# B&R Automation Studio project TD52 (part 142)

#### lGEN2diag.typ
```iecst
TYPE

   DiagActiveBus : STRUCT
        DiagOn : BOOL; (**)
        DiagOnInTransient : BOOL; (**)
        LEANOXErrSettled : BOOL; (**)
        NoTooStrongWGMove : BOOL; (**)
        NoTransient : BOOL; (**)
        NoExtDist : BOOL; (**)
        NoVoltTrans : BOOL; (**)
        GCBMCBsettled : BOOL; (**)
        GridP : BOOL; (**)
        DiagBitmask : DINT; (**)
        NoMinLoad : BOOL; (**)
        TexhSettledAfterRamp : BOOL; (**)
        NoGasMixingTrans : BOOL; (**)
    END_STRUCT;

   tGEN2FDebug : STRUCT
        LambdaCmd : REAL; (*lambda command [-]*)
        y_f : REAL; (*filtered value of y*)
        Residual : REAL; (*high pass filtered lambda (= gradient)*)
        Thrsh : REAL; (*the actual threshold (after scaling)*)
        DiagActive : BOOL; (*diagnosis activated*)
        FaultLambdaOnly : BOOL; (*fault detected based only on lambda gradient (WITHOUT deactivation logic)*)
        ResLambdaOnly : REAL; (*high pass filtered lambda signal (after lambda has been lowpass filtered)*)
        ResLambdaITP : REAL; (*high pass filtered lambda signal due to ITP change (after lambda est. has been lowpass filtered)*)
        ResLambdaEst : REAL; (*high pass filtered estimated lambda signal (after lambda est. has been lowpass filtered)*)
        LambdaEst : REAL; (*estimated lambda (via lookup table) dependent on p2s*)
        LEANOXErr : REAL; (*internally calculated LEANOX error [bar]*)
        TexhAvg : REAL; (*exhaust temperature [°C] (avg.) calculated via the mean value*)
        TexhMin : REAL; (*exhaust temperature [°C] (min.)*)
        GasMixing_RatioHP : REAL; (*high pass filtered gas mixing ratio*)
        DeltaTexhAllowed : REAL; (*max. allowed rise in avg. exhaust temp. [°C] used for fault detection (after scaling)*)
        tDiagActiveBus : DiagActiveBus; (*struct to check which component of the activation logic is on*)
    END_STRUCT;

   tGEN2FIn : STRUCT
        LambdaCmd : REAL; (*lambda command [-]*)
        Lambda_ss : REAL; (*steady state lambda [-]*)
        Reset : BOOL; (*reset of filter blocks*)
        Pset_WR_norm : REAL; (*power reference without a ramp [p.u.]*)
        Pset_norm : REAL; (*power reference trajectory [p.u.]*)
        bExt_dist : BOOL; (*TRUE --> external disturbance*)
        Texh : ARRAY[0..24] OF REAL; (*exhaust temperatures (cylinder specific)*)
        p2s : REAL; (*p2s [bar]*)
        p2sCmd : REAL; (*p2s command (LEANOX) [bar]*)
        posWG_norm : REAL; (*waste-gate position [p.u.] 0...1*)
        WGM_reset : BOOL; (*reset bit for the wastegate monitoring part*)
        LEANOXErrorFiltReset : BOOL; (*reset bit for the lowpass used to filter p2s in the LEANOX error settling detection*)
        bVltg_reset : BOOL; (*reset bit for the voltage monitoring part*)
        U_L1L2_norm : REAL; (*concatenated voltage L1L2 [p.u.]*)
        U_L2L3_norm : REAL; (*concatenated voltage L2L3 [p.u.]*)
        U_L3L1_norm : REAL; (*concatenated voltage L1L2 [p.u.]*)
        Man_Cond_On : BOOL; (*manual override to set the diagnosis to ON*)
        bGCBON : BOOL; (*generator circuit breaker closed information*)
        bMCBON : BOOL; (*main circuit breaker closed information*)
        bPTransDetReset : BOOL; (*reset bit for the transient monitoring part*)
        bAllowDetInTrans : BOOL; (*allow detection during ramps (if LEANOX error is small enough)*)
        bTexhSettled_reset : BOOL; (*reset bit for Texh settled detection (after power ramps)*)
        rGasMixing_Ratio : REAL; (*gas mixing ratio [0 - 100 percent]*)
        bGasMixing_reset : BOOL; (*reset bit for gas mixing settled detection*)
        bFileOnlyInTrans : BOOL; (*write files only during power ramps (only if detection is allowed during ramps)*)
        rITPmean : REAL; (*mean ignition timing point [°CA]*)
    END_STRUCT;

   tGEN2FOut : STRUCT
        FrictionFault : BOOL; (*fault detected based on (negative) lambda gradient and (positive) exh. temp. gradient*)
        FrictionFaultInTransient : BOOL; (*fault detected based on (negative) lambda gradient and (positive) exh. temp. gradient; fault in transient detected (only for writing files at the moment!)*)
    END_STRUCT;

   tGEN2FParameter : STRUCT
        TrshPsetDev : REAL; (*threshold value for power set point deviation [p.u.]*)
        TrshPsetStat : REAL; (*threshold value for steady state detection [p.u.]*)
        TconstPsetStat : REAL; (*timeconstant for steady state detection*)
        TrshLoad : REAL; (*threshold value for load level (related to the set power point) [p.u.]*)
        TConstLP : REAL; (*time constant [s] for the lambda lowpass filter*)
        TConstHP : REAL; (*time constant [s] for the lambda highpass filter (situated after the lowpass)*)
        ITPmeanScaling : REAL; (*scaling for the mean ITP to estimate a lambda change*)
        FaultThrshLambda : REAL; (*threshold value for lambda fault detection*)
        ThrshScale : REAL; (*scaling of the threshold value for lambda fault detection [p.u.]*)
        TPulseLambdaFault : REAL; (*minimum time [s] a lambda fault pulse is provided for further detection (exh. temp.)*)
        NCyl : DINT; (*number of cylinders*)
        DeltaTexhAllowed : REAL; (*max. allowed rise in avg. exhaust temp. used for fault detection*)
        TexhPlausibleMin : REAL; (*min. exhaust temperature which is considered plausible (to exclude faulty sensors)*)
        TexhPlausibleMax : REAL; (*max. exhaust temperature which is considered plausible (to exclude faulty sensors)*)
        WGM_FaultThrsh : REAL; (*wastegate monitoring fault threshold*)
        WGM_Tconst : REAL; (*wastegate monitoring time constant [sec]*)
        LEANOXErrorTconst : REAL; (*time constant [s] for filtering p2s in LEANOX error calculation*)
        LEANOXErrorThrsh : REAL; (*threshold for leanox error (diagnosis gets active if the error is smaller than this threshold)*)
        Vltg_FaultThrsh : REAL; (*voltage monitoring fault threshold*)
        Vltg_Tconst : REAL; (*voltage monitoring time constant [sec]*)
        MonitoringDelay : REAL; (*global monitoring time delay (used for all activation logic pars) [sec]*)
        TexhSettledThrsh : REAL; (*threshold for exhaust temperature settled detection*)
        TexhSettledTConstLP : REAL; (*time constant [s] for the Texh lowpass filter -> settled detection*)
        TexhSettledTConstHP : REAL; (*time constant [s] for the Texh highpass filter (situated after the lowpass) -> settled detection*)
        TexhSettledMaxTD : REAL; (*max. time [s] after a power ramp after which the exhaust temperature is considered settled (even if the filter does not suggest this!)*)
        bGasMixingEnDet : BOOL; (*enable gas mixing transient detection*)
        GasMixingThrsh : REAL; (*threshold for gas mixing transient detection*)
        GasMixingTconstLP : REAL; (*time constant [s] for gas mixing transient detection lowpass*)
        GasMixingTconstHP : REAL; (*time constant [s] for gas mixing transient detection highpass*)
    END_STRUCT;
END_TYPE
TYPE
rtB_TOF_G2Fdiag : STRUCT
	LogicalOperator1 : BOOL;
END_STRUCT;
rtDW_TOF_G2Fdiag : STRUCT
	DiscreteTimeIntegrator_DSTATE : LREAL;
	DiscreteTimeIntegrator_PrevRese : SINT;
	DiscreteTimeIntegrator_IC_LOADI : USINT;
END_STRUCT;
rtB_TON_G2Fdiag : STRUCT
	LogicalOperator3 : BOOL;
END_STRUCT;
rtDW_TON_G2Fdiag : STRUCT
	DiscreteTimeIntegrator_DSTATE : REAL;
	DiscreteTimeIntegrator_PrevRese : SINT;
END_STRUCT;
rtB_TP_G2Fdiag : STRUCT
	Merge : LREAL;
	LogicalOperator1 : BOOL;
END_STRUCT;
rtDW_TP_G2Fdiag : STRUCT
	DelayInput2_DSTATE : LREAL;
	UnitDelay2_DSTATE : BOOL;
END_STRUCT;
BlockIO_G2Fdiag : STRUCT
	BusInput1 : tGEN2FIn;
	BusInput : tGEN2FParameter;
	UnitDelay : UDINT;
	TP1 : rtB_TP_G2Fdiag;
	TP : rtB_TP_G2Fdiag;
	TON_n : rtB_TON_G2Fdiag;
	TON_i : rtB_TON_G2Fdiag;
	TON1 : rtB_TON_G2Fdiag;
	TON_e : rtB_TON_G2Fdiag;
	TOF_o : rtB_TOF_G2Fdiag;
	TOF_h : rtB_TOF_G2Fdiag;
	TON : rtB_TON_G2Fdiag;
	TON_j : rtB_TON_G2Fdiag;
	TON_k : rtB_TON_G2Fdiag;
	TOF : rtB_TOF_G2Fdiag;
END_STRUCT;
D_Work_G2Fdiag : STRUCT
	DiscreteTimeIntegrator_DSTATE : REAL;
	DiscreteTimeIntegrator_DSTATE_k : REAL;
	DiscreteTimeIntegrator_DSTATE_h : REAL;
	DiscreteTimeIntegrator_DSTATE_c : REAL;
	DiscreteTimeIntegrator_DSTATE_p : REAL;
	DiscreteTimeIntegrator_DSTATE_e : REAL;
	DiscreteTimeIntegrator_DSTAT_hv : REAL;
	DiscreteTimeIntegrator_DSTATE_j : REAL;
	DiscreteTimeIntegrator_DSTATE_n : REAL;
	DiscreteTimeIntegrator_DSTATE_o : ARRAY[0..2] OF REAL;
	DiscreteTimeIntegrator_DSTAT_jn : ARRAY[0..2] OF REAL;
	DiscreteTimeIntegrator_DSTATE_a : ARRAY[0..2] OF REAL;
	DiscreteTimeIntegrator_DSTATE_d : ARRAY[0..2] OF REAL;
	DiscreteTimeIntegrator_DSTATE_i : REAL;
	UnitDelay_DSTATE : UDINT;
	Texh_scalar_1 : REAL;
	Texh_min_1 : REAL;
	Texh_scalar_1_f : REAL;
	Texh_min_1_p : REAL;
	DelayInput1_DSTATE : BOOL;
	DelayInput1_DSTATE_e : BOOL;
	DelayInput1_DSTATE_m : BOOL;
	DelayInput1_DSTATE_l : BOOL;
	Delay_DSTATE : BOOL;
	DelayInput1_DSTATE_i : BOOL;
	DelayInput1_DSTATE_n : BOOL;
	DelayInput1_DSTATE_p : BOOL;
	DelayInput1_DSTATE_p3 : BOOL;
	DiscreteTimeIntegrator_PrevRese : SINT;
	DiscreteTimeIntegrator_PrevRe_e : SINT;
	DiscreteTimeIntegrator_PrevRe_j : SINT;
	DiscreteTimeIntegrator_PrevRe_f : SINT;
	DiscreteTimeIntegrator_PrevRe_p : SINT;
	DiscreteTimeIntegrator_PrevR_jm : SINT;
	DiscreteTimeIntegrator_PrevRe_n : SINT;
	DiscreteTimeIntegrator_PrevR_ji : SINT;
	DiscreteTimeIntegrator_PrevR_nv : SINT;
	DiscreteTimeIntegrator_PrevRe_d : SINT;
	DiscreteTimeIntegrator_PrevR_do : SINT;
	DiscreteTimeIntegrator_PrevRe_m : SINT;
	DiscreteTimeIntegrator_PrevRe_a : SINT;
	DiscreteTimeIntegrator_PrevR_ah : SINT;
	DiscreteTimeIntegrator_IC_LOADI : USINT;
	DiscreteTimeIntegrator_IC_LOA_c : USINT;
	DiscreteTimeIntegrator_IC_LOA_b : USINT;
	DiscreteTimeIntegrator_IC_LOA_g : USINT;
	DiscreteTimeIntegrator_IC_LOA_p : USINT;
	DiscreteTimeIntegrator_IC_LOA_o : USINT;
	DiscreteTimeIntegrator_IC_LO_cl : USINT;
	DiscreteTimeIntegrator_IC_LO_ps : USINT;
	DiscreteTimeIntegrator_IC_LOA_h : USINT;
	DiscreteTimeIntegrator_IC_LO_pk : USINT;
	DiscreteTimeIntegrator_IC_LO_c0 : USINT;
	DiscreteTimeIntegrator_IC_LOA_j : USINT;
	DiscreteTimeIntegrator_IC_LOA_e : USINT;
	DiscreteTimeIntegrator_IC_LO_gt : USINT;
	Texh_scalar_1_not_empty : BOOL;
	Texh_scalar_1_not_empty_d : BOOL;
	bSettlingPhase : BOOL;
	TexhSettledAfterRamp_persistent : BOOL;
	TP1 : rtDW_TP_G2Fdiag;
	TP : rtDW_TP_G2Fdiag;
	TON_n : rtDW_TON_G2Fdiag;
	TON_i : rtDW_TON_G2Fdiag;
	TON1 : rtDW_TON_G2Fdiag;
	TON_e : rtDW_TON_G2Fdiag;
	TOF_o : rtDW_TOF_G2Fdiag;
	TOF_h : rtDW_TOF_G2Fdiag;
	TON : rtDW_TON_G2Fdiag;
	TON_j : rtDW_TON_G2Fdiag;
	TON_k : rtDW_TON_G2Fdiag;
	TOF : rtDW_TOF_G2Fdiag;
END_STRUCT;
ExternalInputs_G2Fdiag : STRUCT
	IN : tGEN2FIn;
	para : tGEN2FParameter;
END_STRUCT;
ExternalOutputs_G2Fdiag : STRUCT
	OUT : tGEN2FOut;
	dbg : tGEN2FDebug;
END_STRUCT;
END_TYPE
```

#### G2Fdiag.h
```c
/********************************************************************
 * COPYRIGHT -- Bernecker + Rainer Industrie-Elektronik Ges.m.b.H.
 ********************************************************************
 * Program: G2Fdiag
 * File: G2Fdiag.h
 * Author: 106003773
 * Created: Wed Apr 20 16:09:39 2016
 ********************************************************************
 * Header for program G2Fdiag
 ********************************************************************
 * Generated with B&R Automation Studio Target for Simulink V4.2
 * (ERT based)
 ********************************************************************/

#ifndef RTW_HEADER_G2Fdiag_h_
#define RTW_HEADER_G2Fdiag_h_
#ifndef G2Fdiag_COMMON_INCLUDES_
# define G2Fdiag_COMMON_INCLUDES_
#include <math.h>
#include "rtwtypes.h"
#include "rtw_continuous.h"
#include "rtw_solver.h"
#endif                                 /* G2Fdiag_COMMON_INCLUDES_ */

#include "G2Fdiag_types.h"
#include "lGEN2diag.h"

/* Macros for accessing real-time model data structure */
#ifndef rtmGetErrorStatus
# define rtmGetErrorStatus(rtm)        ((void*) 0)
#endif

#ifndef rtmSetErrorStatus
# define rtmSetErrorStatus(rtm, val)   ((void) 0)
#endif

#ifndef rtmGetStopRequested
# define rtmGetStopRequested(rtm)      ((void*) 0)
#endif

#ifndef MIN
#define MIN(a,b)                       ((a) < (b) ? (a) : (b))
#endif

#ifndef MAX
#define MAX(a,b)                       ((a) > (b) ? (a) : (b))
#endif

/* Block signals for system '<S7>/TOF' */

/* Block states (auto storage) for system '<S7>/TOF' */

/* Block signals for system '<S8>/TON' */

/* Block states (auto storage) for system '<S8>/TON' */

/* Block signals for system '<S6>/TP' */

/* Block states (auto storage) for system '<S6>/TP' */

/* Block signals (auto storage) */

/* Block states (auto storage) for system '<Root>' */

/* External inputs (root inport signals with auto storage) */

/* External outputs (root outports fed by signals with auto storage) */

/* Block signals (auto storage) */
extern BlockIO_G2Fdiag G2Fdiag_B;

/* Block states (auto storage) */
extern D_Work_G2Fdiag G2Fdiag_DWork;

/* External inputs (root inport signals with auto storage) */
extern ExternalInputs_G2Fdiag G2Fdiag_U;

/* External outputs (root outports fed by signals with auto storage) */
extern ExternalOutputs_G2Fdiag G2Fdiag_Y;

/* Model entry point functions */
extern void G2Fdiag_initialize(struct fGEN2diag* inst);
extern void G2Fdiag_step(struct fGEN2diag* inst);
extern void G2Fdiag_terminate(struct fGEN2diag* inst);

/*-
 * The generated code includes comments that allow you to trace directly
 * back to the appropriate location in the model.  The basic format
 * is <system>/block_name, where system is the system number (uniquely
 * assigned by Simulink) and block_name is the name of the block.
 *
 * Use the MATLAB hilite_system command to trace the generated code back
 * to the model.  For example,
 *
 * hilite_system('<S3>')    - opens system 3
 * hilite_system('<S3>/Kp') - opens and selects block Kp which resides in S3
 *
 * Here is the system hierarchy for this model
 *
 * '<Root>' : 'G2Fdiag'
 * '<S1>'   : 'G2Fdiag/Environment Controller'
 * '<S2>'   : 'G2Fdiag/Environment Controller1'
 * '<S3>'   : 'G2Fdiag/GEN2_Friction_Detection'
 * '<S4>'   : 'G2Fdiag/Info'
 * '<S5>'   : 'G2Fdiag/GEN2_Friction_Detection/DiagActivLogic'
 * '<S6>'   : 'G2Fdiag/GEN2_Friction_Detection/Fault Detection'
 * '<S7>'   : 'G2Fdiag/GEN2_Friction_Detection/DiagActivLogic/Exteternal disturbance'
 * '<S8>'   : 'G2Fdiag/GEN2_Friction_Detection/DiagActivLogic/GBC and MBC monitoring'
 * '<S9>'   : 'G2Fdiag/GEN2_Friction_Detection/DiagActivLogic/GasMixingTransient'
 * '<S10>'  : 'G2Fdiag/GEN2_Friction_Detection/DiagActivLogic/LEANOX error monitoring'
 * '<S11>'  : 'G2Fdiag/GEN2_Friction_Detection/DiagActivLogic/Min Load Detection'
 * '<S12>'  : 'G2Fdiag/GEN2_Friction_Detection/DiagActivLogic/Power ramp detection'
 * '<S13>'  : 'G2Fdiag/GEN2_Friction_Detection/DiagActivLogic/Texh settled after power ramp'
 * '<S14>'  : 'G2Fdiag/GEN2_Friction_Detection/DiagActivLogic/Voltage monitoring'
 * '<S15>'  : 'G2Fdiag/GEN2_Friction_Detection/DiagActivLogic/Wastegate monitoring'
 * '<S16>'  : 'G2Fdiag/GEN2_Friction_Detection/DiagActivLogic/Exteternal disturbance/TOF'
 * '<S17>'  : 'G2Fdiag/GEN2_Friction_Detection/DiagActivLogic/Exteternal disturbance/TOF/Data Type Conversion Inherited'
 * '<S18>'  : 'G2Fdiag/GEN2_Friction_Detection/DiagActivLogic/GBC and MBC monitoring/State Change GCB'
 * '<S19>'  : 'G2Fdiag/GEN2_Friction_Detection/DiagActivLogic/GBC and MBC monitoring/State Change MCB'
 * '<S20>'  : 'G2Fdiag/GEN2_Friction_Detection/DiagActivLogic/GBC and MBC monitoring/TON'
 * '<S21>'  : 'G2Fdiag/GEN2_Friction_Detection/DiagActivLogic/GBC and MBC monitoring/State Change GCB/Detect Fall Nonpositive'
 * '<S22>'  : 'G2Fdiag/GEN2_Friction_Detection/DiagActivLogic/GBC and MBC monitoring/State Change GCB/Detect Rise Positive'
 * '<S23>'  : 'G2Fdiag/GEN2_Friction_Detection/DiagActivLogic/GBC and MBC monitoring/State Change GCB/Detect Fall Nonpositive/Nonpositive'
 * '<S24>'  : 'G2Fdiag/GEN2_Friction_Detection/DiagActivLogic/GBC and MBC monitoring/State Change GCB/Detect Rise Positive/Positive'
 * '<S25>'  : 'G2Fdiag/GEN2_Friction_Detection/DiagActivLogic/GBC and MBC monitoring/State Change MCB/Detect Fall Nonpositive'
 * '<S26>'  : 'G2Fdiag/GEN2_Friction_Detection/DiagActivLogic/GBC and MBC monitoring/State Change MCB/Detect Rise Positive'
 * '<S27>'  : 'G2Fdiag/GEN2_Friction_Detection/DiagActivLogic/GBC and MBC monitoring/State Change MCB/Detect Fall Nonpositive/Nonpositive'
 * '<S28>'  : 'G2Fdiag/GEN2_Friction_Detection/DiagActivLogic/GBC and MBC monitoring/State Change MCB/Detect Rise Positive/Positive'
 * '<S29>'  : 'G2Fdiag/GEN2_Friction_Detection/DiagActivLogic/GBC and MBC monitoring/TON/Data Type Conversion Inherited'
 * '<S30>'  : 'G2Fdiag/GEN2_Friction_Detection/DiagActivLogic/GasMixingTransient/TON'
 * '<S31>'  : 'G2Fdiag/GEN2_Friction_Detection/DiagActivLogic/GasMixingTransient/filterTexh'
 * '<S32>'  : 'G2Fdiag/GEN2_Friction_Detection/DiagActivLogic/GasMixingTransient/highpass gas mixing'
 * '<S33>'  : 'G2Fdiag/GEN2_Friction_Detection/DiagActivLogic/GasMixingTransient/TON/Data Type Conversion Inherited'
 * '<S34>'  : 'G2Fdiag/GEN2_Friction_Detection/DiagActivLogic/GasMixingTransient/highpass gas mixing/filter4'
 * '<S35>'  : 'G2Fdiag/GEN2_Friction_Detection/DiagActivLogic/LEANOX error monitoring/TON'
 * '<S36>'  : 'G2Fdiag/GEN2_Friction_Detection/DiagActivLogic/LEANOX error monitoring/filter4'
 * '<S37>'  : 'G2Fdiag/GEN2_Friction_Detection/DiagActivLogic/LEANOX error monitoring/TON/Data Type Conversion Inherited'
 * '<S38>'  : 'G2Fdiag/GEN2_Friction_Detection/DiagActivLogic/Min Load Detection/TOF'
 * '<S39>'  : 'G2Fdiag/GEN2_Friction_Detection/DiagActivLogic/Min Load Detection/TOF/Data Type Conversion Inherited'
 * '<S40>'  : 'G2Fdiag/GEN2_Friction_Detection/DiagActivLogic/Power ramp detection/TOF'
 * '<S41>'  : 'G2Fdiag/GEN2_Friction_Detection/DiagActivLogic/Power ramp detection/filter4'
 * '<S42>'  : 'G2Fdiag/GEN2_Friction_Detection/DiagActivLogic/Power ramp detection/TOF/Data Type Conversion Inherited'
 * '<S43>'  : 'G2Fdiag/GEN2_Friction_Detection/DiagActivLogic/Texh settled after power ramp/Detect Fall Nonpositive'
 * '<S44>'  : 'G2Fdiag/GEN2_Friction_Detection/DiagActivLogic/Texh settled after power ramp/Detect Rise Positive'
 * '<S45>'  : 'G2Fdiag/GEN2_Friction_Detection/DiagActivLogic/Texh settled after power ramp/MATLAB Function'
 * '<S46>'  : 'G2Fdiag/GEN2_Friction_Detection/DiagActivLogic/Texh settled after power ramp/TON'
 * '<S47>'  : 'G2Fdiag/GEN2_Friction_Detection/DiagActivLogic/Texh settled after power ramp/TON1'
 * '<S48>'  : 'G2Fdiag/GEN2_Friction_Detection/DiagActivLogic/Texh settled after power ramp/filterTexh'
 * '<S49>'  : 'G2Fdiag/GEN2_Friction_Detection/DiagActivLogic/Texh settled after power ramp/highpassTexh'
 * '<S50>'  : 'G2Fdiag/GEN2_Friction_Detection/DiagActivLogic/Texh settled after power ramp/Detect Fall Nonpositive/Nonpositive'
 * '<S51>'  : 'G2Fdiag/GEN2_Friction_Detection/DiagActivLogic/Texh settled after power ramp/Detect Rise Positive/Positive'
 * '<S52>'  : 'G2Fdiag/GEN2_Friction_Detection/DiagActivLogic/Texh settled after power ramp/TON/Data Type Conversion Inherited'
 * '<S53>'  : 'G2Fdiag/GEN2_Friction_Detection/DiagActivLogic/Texh settled after power ramp/TON1/Data Type Conversion Inherited'
 * '<S54>'  : 'G2Fdiag/GEN2_Friction_Detection/DiagActivLogic/Texh settled after power ramp/highpassTexh/filter4'
 * '<S55>'  : 'G2Fdiag/GEN2_Friction_Detection/DiagActivLogic/Voltage monitoring/TON'
 * '<S56>'  : 'G2Fdiag/GEN2_Friction_Detection/DiagActivLogic/Voltage monitoring/voltage phase 1'
 * '<S57>'  : 'G2Fdiag/GEN2_Friction_Detection/DiagActivLogic/Voltage monitoring/voltage phase 2'
 * '<S58>'  : 'G2Fdiag/GEN2_Friction_Detection/DiagActivLogic/Voltage monitoring/voltage phase 3'
 * '<S59>'  : 'G2Fdiag/GEN2_Friction_Detection/DiagActivLogic/Voltage monitoring/TON/Data Type Conversion Inherited'
 * '<S60>'  : 'G2Fdiag/GEN2_Friction_Detection/DiagActivLogic/Voltage monitoring/voltage phase 1/filter4'
 * '<S61>'  : 'G2Fdiag/GEN2_Friction_Detection/DiagActivLogic/Voltage monitoring/voltage phase 2/filter4'
 * '<S62>'  : 'G2Fdiag/GEN2_Friction_Detection/DiagActivLogic/Voltage monitoring/voltage phase 3/filter4'
 * '<S63>'  : 'G2Fdiag/GEN2_Friction_Detection/DiagActivLogic/Wastegate monitoring/TON'
 * '<S64>'  : 'G2Fdiag/GEN2_Friction_Detection/DiagActivLogic/Wastegate monitoring/filter4'
 * '<S65>'  : 'G2Fdiag/GEN2_Friction_Detection/DiagActivLogic/Wastegate monitoring/TON/Data Type Conversion Inherited'
 * '<S66>'  : 'G2Fdiag/GEN2_Friction_Detection/Fault Detection/Detect Increase'
 * '<S67>'  : 'G2Fdiag/GEN2_Friction_Detection/Fault Detection/Detect Increase1'
 * '<S68>'  : 'G2Fdiag/GEN2_Friction_Detection/Fault Detection/TP'
 * '<S69>'  : 'G2Fdiag/GEN2_Friction_Detection/Fault Detection/TP1'
 * '<S70>'  : 'G2Fdiag/GEN2_Friction_Detection/Fault Detection/detection logic'
 * '<S71>'  : 'G2Fdiag/GEN2_Friction_Detection/Fault Detection/detection logic1'
 * '<S72>'  : 'G2Fdiag/GEN2_Friction_Detection/Fault Detection/highpass1'
 * '<S73>'  : 'G2Fdiag/GEN2_Friction_Detection/Fault Detection/highpass2'
 * '<S74>'  : 'G2Fdiag/GEN2_Friction_Detection/Fault Detection/lowpass1'
 * '<S75>'  : 'G2Fdiag/GEN2_Friction_Detection/Fault Detection/lowpass2'
 * '<S76>'  : 'G2Fdiag/GEN2_Friction_Detection/Fault Detection/vector to scalar (mean, etc.)'
 * '<S77>'  : 'G2Fdiag/GEN2_Friction_Detection/Fault Detection/TP/Compare To Zero'
 * '<S78>'  : 'G2Fdiag/GEN2_Friction_Detection/Fault Detection/TP/Enabled Subsystem'
 * '<S79>'  : 'G2Fdiag/GEN2_Friction_Detection/Fault Detection/TP/Enabled Subsystem1'
 * '<S80>'  : 'G2Fdiag/GEN2_Friction_Detection/Fault Detection/TP/Rate Limiter'
 * '<S81>'  : 'G2Fdiag/GEN2_Friction_Detection/Fault Detection/TP/Rate Limiter/Saturation Dynamic'
 * '<S82>'  : 'G2Fdiag/GEN2_Friction_Detection/Fault Detection/TP1/Compare To Zero'
 * '<S83>'  : 'G2Fdiag/GEN2_Friction_Detection/Fault Detection/TP1/Enabled Subsystem'
 * '<S84>'  : 'G2Fdiag/GEN2_Friction_Detection/Fault Detection/TP1/Enabled Subsystem1'
 * '<S85>'  : 'G2Fdiag/GEN2_Friction_Detection/Fault Detection/TP1/Rate Limiter'
 * '<S86>'  : 'G2Fdiag/GEN2_Friction_Detection/Fault Detection/TP1/Rate Limiter/Saturation Dynamic'
 * '<S87>'  : 'G2Fdiag/GEN2_Friction_Detection/Fault Detection/highpass1/filter4'
 * '<S88>'  : 'G2Fdiag/GEN2_Friction_Detection/Fault Detection/highpass2/filter4'
 */
#endif                                 /* RTW_HEADER_G2Fdiag_h_ */
```

#### G2Fdiag_private.h
```c
/********************************************************************
 * COPYRIGHT -- Bernecker + Rainer Industrie-Elektronik Ges.m.b.H.
 ********************************************************************
 * Program: G2Fdiag
 * File: G2Fdiag_private.h
 * Author: 106003773
 * Created: Wed Apr 20 16:09:39 2016
 ********************************************************************
 * Header for program G2Fdiag
 ********************************************************************
 * Generated with B&R Automation Studio Target for Simulink V4.2
 * (ERT based)
 ********************************************************************/

#ifndef RTW_HEADER_G2Fdiag_private_h_
#define RTW_HEADER_G2Fdiag_private_h_
#include "rtwtypes.h"
#include <bur/plctypes.h>
#ifndef __RTWTYPES_H__
#error This file requires rtwtypes.h to be included
#else
#ifdef TMWTYPES_PREVIOUSLY_INCLUDED
#error This file requires rtwtypes.h to be included before tmwtypes.h
#else

/* Check for inclusion of an incorrect version of rtwtypes.h */
#ifndef RTWTYPES_ID_C08S16I32L32N32F1
#error This code was generated with a different "rtwtypes.h" than the file included
#endif                                 /* RTWTYPES_ID_C08S16I32L32N32F1 */
#endif                                 /* TMWTYPES_PREVIOUSLY_INCLUDED */
#endif                                 /* __RTWTYPES_H__ */

#ifndef MIN
#define MIN(a,b)                       ((a) < (b) ? (a) : (b))
#endif

#ifndef MAX
#define MAX(a,b)                       ((a) > (b) ? (a) : (b))
#endif

extern void G2Fdiag_TOF_Init(rtDW_TOF_G2Fdiag *localDW, struct fGEN2diag* inst);
extern void G2Fdiag_TOF(boolean_T rtu_IN, real_T rtu_PT, rtB_TOF_G2Fdiag *localB,
  rtDW_TOF_G2Fdiag *localDW, struct fGEN2diag* inst);
extern void G2Fdiag_TON(boolean_T rtu_IN, real32_T rtu_PT, rtB_TON_G2Fdiag
  *localB, rtDW_TON_G2Fdiag *localDW, struct fGEN2diag* inst);
extern void G2Fdiag_EnabledSubsystem(boolean_T rtu_0, real_T rtu_1, real_T
  *rty_Out1, struct fGEN2diag* inst);
extern void G2Fdiag_TP_Init(rtDW_TP_G2Fdiag *localDW, struct fGEN2diag* inst);
extern void G2Fdiag_TP(boolean_T rtu_IN, real_T rtu_PT, rtB_TP_G2Fdiag *localB,
  rtDW_TP_G2Fdiag *localDW, struct fGEN2diag* inst);

#endif                                 /* RTW_HEADER_G2Fdiag_private_h_ */
```

#### G2Fdiag_types.h
```c
/********************************************************************
 * COPYRIGHT -- Bernecker + Rainer Industrie-Elektronik Ges.m.b.H.
 ********************************************************************
 * Program: G2Fdiag
 * File: G2Fdiag_types.h
 * Author: 106003773
 * Created: Wed Apr 20 16:09:39 2016
 ********************************************************************
 * Header for program G2Fdiag
 ********************************************************************
 * Generated with B&R Automation Studio Target for Simulink V4.2
 * (ERT based)
 ********************************************************************/

#ifndef RTW_HEADER_G2Fdiag_types_h_
#define RTW_HEADER_G2Fdiag_types_h_
#include "rtwtypes.h"
#ifndef MIN
#define MIN(a,b)                       ((a) < (b) ? (a) : (b))
#endif

#ifndef MAX
#define MAX(a,b)                       ((a) > (b) ? (a) : (b))
#endif

#endif                                 /* RTW_HEADER_G2Fdiag_types_h_ */
```

#### rtwtypes.h
```c
/********************************************************************
 * COPYRIGHT -- Bernecker + Rainer Industrie-Elektronik Ges.m.b.H.
 ********************************************************************
 * Program: G2Fdiag
 * File: rtwtypes.h
 * Author: 106003773
 * Created: Wed Apr 20 16:09:39 2016
 ********************************************************************
 * Header for program G2Fdiag
 ********************************************************************
 * Generated with B&R Automation Studio Target for Simulink V4.2
 * (ERT based)
 ********************************************************************/

#ifndef __RTWTYPES_H__
#define __RTWTYPES_H__
#ifndef TRUE
# define TRUE                          (1U)
#endif

#ifndef FALSE
# define FALSE                         (0U)
#endif

#ifndef __TMWTYPES__
#define __TMWTYPES__
#include <limits.h>

/*=======================================================================*
 * Target hardware information
 *   Device type: Intel->x86/Pentium
 *   Number of bits:     char:   8    short:   16    long:  32
 *                       long:  32
 *                       native word size:  32
 *   Byte ordering: LittleEndian
 *   Signed integer division rounds to: Zero
 *   Shift right on a signed integer as arithmetic shift: on
 *=======================================================================*/

/*=======================================================================*
 * Fixed width word size data types:                                     *
 *   int8_T, int16_T, int32_T     - signed 8, 16, or 32 bit integers     *
 *   uint8_T, uint16_T, uint32_T  - unsigned 8, 16, or 32 bit integers   *
 *   real32_T, real64_T           - 32 and 64 bit floating point numbers *
 *=======================================================================*/
typedef signed char int8_T;
typedef unsigned char uint8_T;
typedef short int16_T;
typedef unsigned short uint16_T;
typedef long int32_T;
typedef unsigned long uint32_T;
typedef float real32_T;
typedef double real64_T;

/*===========================================================================*
 * Generic type definitions: real_T, time_T, boolean_T, int_T, uint_T,       *
 *                           ulong_T, char_T and byte_T.                     *
 *===========================================================================*/
typedef double real_T;
typedef double time_T;
typedef unsigned char boolean_T;
typedef long int_T;
typedef unsigned long uint_T;
typedef unsigned long ulong_T;
typedef char char_T;
typedef unsigned char uchar_T;
typedef char_T byte_T;

/*=======================================================================*
 * Min and Max:                                                          *
 *   int8_T, int16_T, int32_T     - signed 8, 16, or 32 bit integers     *
 *   uint8_T, uint16_T, uint32_T  - unsigned 8, 16, or 32 bit integers   *
 *=======================================================================*/
#define MAX_int8_T                     ((int8_T)(127))
#define MIN_int8_T                     ((int8_T)(-128))
#define MAX_uint8_T                    ((uint8_T)(255U))
#define MIN_uint8_T                    ((uint8_T)(0U))
#define MAX_int16_T                    ((int16_T)(32767))
#define MIN_int16_T                    ((int16_T)(-32768))
#define MAX_uint16_T                   ((uint16_T)(65535U))
#define MIN_uint16_T                   ((uint16_T)(0U))
#define MAX_int32_T                    ((int32_T)(2147483647))
#define MIN_int32_T                    ((int32_T)(-2147483647-1))
#define MAX_uint32_T                   ((uint32_T)(0xFFFFFFFFU))
#define MIN_uint32_T                   ((uint32_T)(0U))

/* Logical type definitions */
#if (!defined(__cplusplus)) && (!defined(__true_false_are_keywords))
#  ifndef false
#   define false                       (0U)
#  endif

#  ifndef true
#   define true                        (1U)
#  endif
#endif

/*
 * Simulink Coder assumes the code is compiled on a target using a 2's complement representation
 * for signed integer values.
 */
#if ((SCHAR_MIN + 1) != -SCHAR_MAX)
#error "This code must be compiled using a 2's complement representation for signed integer values"
#endif

/* This ID is used to detect inclusion of an incompatible rtwtypes.h */
#define RTWTYPES_ID_C08S16I32L32N32F1
#else                                  /* __TMWTYPES__ */
#define TMWTYPES_PREVIOUSLY_INCLUDED
#endif                                 /* __TMWTYPES__ */

/* Block D-Work pointer type */
typedef void * pointer_T;

/* Simulink specific types */
#ifndef __SIMSTRUC_TYPES_H__
#define __SIMSTRUC_TYPES_H__

/* Trigger directions: falling, either, and rising */
typedef enum {
  FALLING_ZERO_CROSSING = -1,
  ANY_ZERO_CROSSING = 0,
  RISING_ZERO_CROSSING = 1
} ZCDirection;

/* Previous state of a trigger signal */
typedef uint8_T ZCSigState;

/* Initial value of a trigger zero crossing signal */
#define UNINITIALIZED_ZCSIG            0x03U
#define NEG_ZCSIG                      0x02U
#define POS_ZCSIG                      0x01U
#define ZERO_ZCSIG                     0x00U

/* Current state of a trigger signal */
typedef enum {
  FALLING_ZCEVENT = -1,
  NO_ZCEVENT = 0,
  RISING_ZCEVENT = 1
} ZCEventType;

#endif                                 /* __SIMSTRUC_TYPES_H__ */
#endif                                 /* __RTWTYPES_H__ */

#ifndef MIN
#define MIN(a,b)                       ((a) < (b) ? (a) : (b))
#endif

#ifndef MAX
#define MAX(a,b)                       ((a) > (b) ? (a) : (b))
#endif
```
